(* PLC project Unnamed, Unknown Unnamed 1 *)
(* stored: creationDateTime 2023-01-25T13:19:30, modificationDateTime 2023-01-25T21:28:01 *)

PROGRAM main
  VAR
    Conveyor AT %QX100.0 : BOOL;
    Prox AT %IX100.0 : BOOL;
    StartButton AT %IX100.1 : BOOL;
  END_VAR

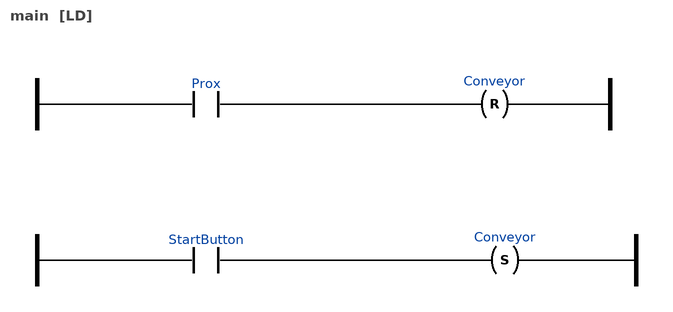
(* LD diagram, written out as Structured Text *)
IF Prox THEN Conveyor := FALSE; END_IF;
IF StartButton THEN Conveyor := TRUE; END_IF;
END_PROGRAM

CONFIGURATION Config0
  RESOURCE Res0 ON PLC
    TASK task0(INTERVAL := T#20ms, PRIORITY := 0);
    PROGRAM instance0 WITH task0 : main;
  END_RESOURCE
END_CONFIGURATION
